// TIA Portal V16 export
// export: Created 2021-11-12T13:32:38.6981798Z, ExportSetting WithDefaults, DisplayName Totally Integrated Automation Portal, DisplayVersion V16 Update 3, DisplayName TIA Portal Version Control Interface, DisplayVersion V16 Update 2, DisplayName TIA Portal Openness, DisplayVersion V16 Update 3, DisplayName SINAMICS Startdrive Advanced, DisplayVersion V16 Update 5, DisplayName SINAMICS Startdrive G130, G150, S120, S150, SINAMICS MV, S210, DisplayVersion V16 Update 5, DisplayName SINAMICS Startdrive G110M, G120, G120C, G120D, G120P, G115D, DisplayVersion V16 Update 5, DisplayName STEP 7 Professional, DisplayVersion V16 Update 3, DisplayName STEP 7 Safety, DisplayVersion V16, DisplayName WinCC UA Professional, DisplayVersion V16 Update 3
DATA_BLOCK "HMI_CMD_2R1"   // DB41
{ S7_Optimized_Access := 'TRUE' }
VERSION : 0.1
// stored: AutoNumber true, DBAccessibleFromOPCUA true, IsOnlyStoredInLoadMemory false, IsRetainMemResEnabled false, IsWriteProtectedInAS false, MemoryReserve 100
   VAR
      xxxxx___BinarySensors___xxxxx_1 : Byte;
      "CM01-BL01_4" : "UDT_CH_DI_Command";   // Proplachovací nádrž 1 Vysoká hladina Varování
      "CM01-BL01_5" : "UDT_CH_DI_Command";   // Proplachovací nádrž 1 Vysoká hladina Max
      xxxxx___BinaryOthers___xxxxx_1 : Byte;
      PwrOK : "UDT_CH_DI_Command";
      "000UH11-SF12" : "UDT_CH_DI_Command";   // Okamžitý stop Robot 2R1
      "000+UH10-SF30" : "UDT_CH_DI_Command";   // Okamžitý stop Robot 2R1, 2R2
      "000UH11-SF08" : "UDT_CH_DI_Command";   // Robot 2R1 Proplach
      "000UH11-SF09" : "UDT_CH_DI_Command";   // Robot 2R1 Nástřik
      RO01_ReqToolchange : Bool;   // Go to position for change tool request
      xxxxx___AnalogueSensors___xxxxx_1 : Byte;
      xxxxx___Drives___xxxxx_1 : Byte;
      RO01 : "UDT_RobotABB_Command";   // Robot
      RC01 : "UDT_DriveRobotABB_Command";   // Controller
      xxxxx___Others___xxxxx_1 : Byte;
      FlushToolCmd : Bool;   // Command to flush tool
      FlushToolEnable : Bool;   // Enable flush tool after end of production
      xxxxx__Alarms___xxxxx : Byte;
      RO01_Timeout : "UDT_DI_Mon_Command";   // Robot job active for too long
      RO01_LubStartErr : "UDT_DI_Mon_Command";   // Lubrication job did not start (robot did not move)
      MixSysErr : "UDT_DI_Mon_Command";   // Mixing system error
      "CM01-BL01_4_alarm" : "UDT_DI_Mon_Command";   // Proplachovací nádrž 1 Vysoká hladina Varování
      "CM01-BL01_5_alarm" : "UDT_DI_Mon_Command";   // Proplachovací nádrž 1 Vysoká hladina Max
      xxxxx___SftyAlarms___xxxxx_1 : Byte;
      ES : "UDT_DI_Mon_Command";   // E-stop
   END_VAR
BEGIN
END_DATA_BLOCK
